(* CODESYS project Device.export

Project tree, tasks and I/O mapping:
  Device : CODESYS Control Win V3, 3S - Smart Software Solutions GmbH, version 3.5.16.0
    application Application
      libraries: Standard, * (System)
      task MainTask (cyclic, interval t#20ms, priority 1) calls PLC_PRG
      task VISU_TASK (cyclic, interval 100 ms, priority 31) calls VisuElems.Visu_Prg
      global variables Globale_Variablen
      program PLC_PRG [FBD]
      function block POU_Abbruch [ST]
      function block POU_Admin [ST]
      function block POU_Auswahltaste [ST]
      function block POU_Becheranzeige [FBD]
      function block POU_BecheranzeigeAuto [ST]
      function block POU_BecheranzeigeManuel [ST]
      function block POU_Kaffee_oder_Tee [ST]
      function block POU_KundenZaehler [ST]
      visualisation Visualisierung_Getrankeautomat
*)

// Device/Application/Globale_Variablen
{attribute 'qualified_only'}
VAR_GLOBAL
	// Variable für die Simulation der Becheranzeige
	Fuellstand: INT := 0;
	Leer: BOOL;
	Full: BOOL;
	// Eingänge
	S1:BOOL; // Kaffee
	S2:BOOL; // Tee
	S3:BOOL; // Zucker
	S4:BOOL; // Milch
	S5:BOOL; // Münzeinwurf
	S6:BOOL; // Admin
	S9:BOOL; // Abbruch
	// Anzeigen
	H1:BOOL; // Kaffee
	H2:BOOL;// Tee
	H3:INT := 0; // Zucker
	H4:INT := 0; // Milch
	H5:BOOL; // Münzeinwurf
	H6:BOOL; // Admin
	H9: BOOL ; // Abbruch
	// Variable für die "Kundenzähler"
	KundenZahl:Word;
	disp_Kundenzahl:STRING;
	// Displayvariable
	Display:STRING;
	//Verriegelungsvariablen für Milch und Zucker
	Flanke1:BOOL:=TRUE;
	Flanke2:BOOL:=TRUE;
	G1:BOOL:=TRUE;
	G2:BOOL:=True;
	// Füllsensor 
	HB2:BOOL;
	B2:BOOL;
	B1:BOOL;
	// 
	x2:BOOL;
	K1:BOOL:=TRUE;
	
	// Variable für die Dosierung Milch und Zucker
	Anzahl1:INT;
    Anzahl2:INT;
END_VAR

// Device/Application/PLC_PRG
PROGRAM PLC_PRG
VAR
	
	
	// abgelaufende Zeit
	Zeit: TIME;
	Zeitint: INT := 0;
	
	POU_Becheranzeige: POU_Becheranzeige;
	
	//POU_Kaffee_0: POU_Kaffee;
	//POU_Tee_0: POU_Tee;
	

	POU_0: POU_Kaffee_oder_Tee;
	POU_Abbruch_0: POU_Abbruch;
	POU_Becheranzeige_0: POU_Becheranzeige;
	POU_Auswahltaste_0: POU_Auswahltaste;
	POU_Admin_0: POU_Admin;
	POU_KundenZahl_0: POU_KundenZaehler;
	POU_BecheranzeigeAuto_0: POU_BecheranzeigeAuto;
	POU_BecheranzeigeManuel_0: POU_BecheranzeigeManuel;
	

END_VAR

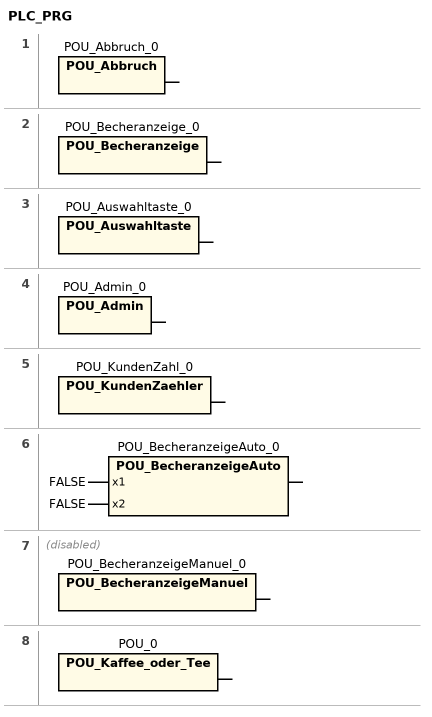
// NETWORK 1
POU_Abbruch_0(); // POU_Abbruch

// NETWORK 2
POU_Becheranzeige_0(); // POU_Becheranzeige

// NETWORK 3
POU_Auswahltaste_0(); // POU_Auswahltaste

// NETWORK 4
POU_Admin_0(); // POU_Admin

// NETWORK 5
POU_KundenZahl_0(); // POU_KundenZaehler

// NETWORK 6
POU_BecheranzeigeAuto_0(x1 := FALSE, x2 := FALSE); // POU_BecheranzeigeAuto

// NETWORK 7 (disabled)
// POU_BecheranzeigeManuel_0(); // POU_BecheranzeigeManuel

// NETWORK 8
POU_0(); // POU_Kaffee_oder_Tee

END_PROGRAM

// Device/Application/POU_Abbruch
FUNCTION_BLOCK POU_Abbruch
VAR_INPUT
END_VAR
VAR_OUTPUT
END_VAR
VAR
END_VAR

Globale_Variablen.H9:= Globale_Variablen.S9;
IF (Globale_Variablen.H9  = TRUE AND Globale_Variablen.Leer = FALSE AND Globale_Variablen.B1=FALSE )THEN
	
	Globale_Variablen.K1 := TRUE;
	Globale_Variablen.S1:= FALSE;
	Globale_Variablen.S2:= FALSE;
	Globale_Variablen.H1:= FALSE;
	Globale_Variablen.H2:= FALSE;
//Globale_Variablen.S3:= FALSE;
 //	Globale_Variablen.S4:= FALSE;
	Globale_Variablen.H3:= 0;
	Globale_Variablen.H4:= 0;
	Globale_Variablen.H5:= FALSE;
	Globale_Variablen.S5:= FALSE;
	//Globale_Variablen.H6:= FALSE;
	//Globale_Variablen.S6:= FALSE;
	Globale_Variablen.Display := 'Abbruch';
	//Globale_Variablen.H9:= TRUE;
	Globale_Variablen.Leer:=FALSE;
	Globale_Variablen.Full:=FALSE;
	Globale_Variablen.G1 := TRUE;
	
END_IF
// In der oberen If Bedingung wird gefragt ob die Abbruchtaster S9 betätig wurde , wenn ja 
// dann soll alles abgebrochen werden und Lampe H9 leuchten so lange S9 betätigt ist . 

IF Globale_Variablen.H9=FALSE THEN
		//Globale_Variablen.H9:= FALSE;
		Globale_Variablen.Display := 'Bereit';
END_IF

END_FUNCTION_BLOCK

// Device/Application/POU_Becheranzeige
FUNCTION_BLOCK POU_Becheranzeige

VAR	
	//Fuellstand: INT := 0;
	//Leer: BOOL;
	//Voll: BOOL;
END_VAR

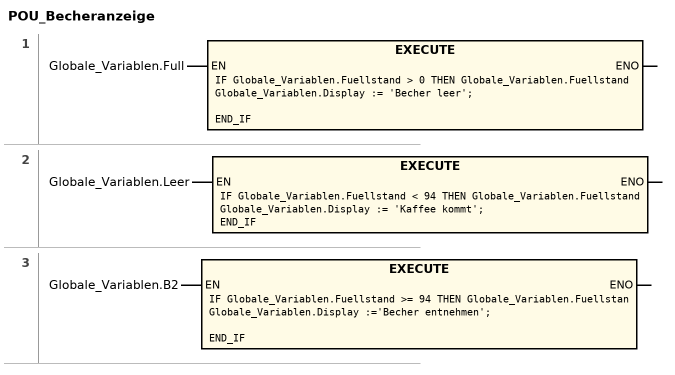
// NETWORK 1
IF Globale_Variablen.Full THEN
    IF Globale_Variablen.Fuellstand > 0 THEN Globale_Variablen.Fuellstand := 0;
    Globale_Variablen.Display := 'Becher leer';
    
    END_IF
END_IF

// NETWORK 2
IF Globale_Variablen.Leer THEN
    IF Globale_Variablen.Fuellstand < 94 THEN Globale_Variablen.Fuellstand := Globale_Variablen.Fuellstand + 1;
    Globale_Variablen.Display := 'Kaffee kommt';
    END_IF
END_IF

// NETWORK 3
IF Globale_Variablen.B2 THEN
    IF Globale_Variablen.Fuellstand >= 94 THEN Globale_Variablen.Fuellstand := 0;
    Globale_Variablen.Display :='Becher entnehmen';
    	
    END_IF
END_IF

END_FUNCTION_BLOCK

// Device/Application/POU_Auswahltaste
FUNCTION_BLOCK POU_Auswahltaste
VAR_INPUT
END_VAR
VAR_OUTPUT
END_VAR
VAR
Merker1:BOOL;
Anzahl3:INT;
Merker2:BOOL;
Anzahl4:INT;


END_VAR

// H3 Zuckeranzeige

Globale_Variablen.Flanke1 := Globale_Variablen.S3 AND NOT Merker1 ;
Merker1 := Globale_Variablen.S3;

IF Globale_Variablen.Flanke1 = 1 AND Globale_Variablen.G1=TRUE THEN 
	Anzahl3 :=Anzahl3 +1;
	Globale_Variablen.H3:=Anzahl3;
END_IF


IF Merker1 = TRUE  THEN 

IF Anzahl3 <= 3 THEN
	CASE Anzahl3 OF
      
		1: Globale_Variablen.Display := '1x Zucker'; 
		2:  Globale_Variablen.Display := '2x Zucker';
		ELSE 
			Globale_Variablen.H3 := 0;
			
 	END_CASE


END_IF
END_IF

IF (Anzahl3 >= 3 OR  Globale_Variablen.S9) THEN
	Anzahl3 := 0;
END_IF

// H4 Milchanzeige
Globale_Variablen.Flanke2 := Globale_Variablen.S4 AND NOT Merker2 AND Globale_Variablen.G1;
Merker2 := Globale_Variablen.S4;


IF Globale_Variablen.Flanke2 = 1 AND Globale_Variablen.G2=TRUE THEN 
	Anzahl4 :=Anzahl4 +1;
	Globale_Variablen.H4:=Anzahl4;
END_IF


IF Merker2 =TRUE  THEN 

IF Anzahl4 <= 3 THEN
	CASE Anzahl4 OF
      
		1: Globale_Variablen.Display := '1x Milch'; 
		2:  Globale_Variablen.Display := '2x Milch';
		ELSE 
			Globale_Variablen.H4 := 0;
			
 	END_CASE
		
END_IF
END_IF

IF (Anzahl4 >= 3 OR    Globale_Variablen.S9) THEN
	Anzahl4 := 0;
END_IF


IF (Anzahl3 >= 3 OR    Globale_Variablen.S9) THEN
	Anzahl3 := 0;
END_IF

END_FUNCTION_BLOCK

// Device/Application/POU_Admin
FUNCTION_BLOCK POU_Admin
VAR_INPUT
END_VAR
VAR_OUTPUT
END_VAR
VAR
I:INT;
x1:Bool;
Flanke1:BOOL;
Flanke2:BOOL;
Merker1:BOOL;
Merker2:BOOL;
MerkerS6:BOOL;
Merker3:BOOL;
Merker4:BOOL;
MerkerS5:BOOL;

Anzahl1:INT;
Anzahl2:INT;
END_VAR

// Globale_Variablen.H6 :=Globale_Variablen.S6;
// IF Globale_Variablen.H6 = TRUE THEN 
// 
// END_IF 
Merker3:=Globale_Variablen.H5;
 
// die Lokale Variable Merker3 dient dazu , ob die Taster S5 betätigt ist  und dementsprechend H5 leuchtet
// wenn ja , dann soll der Programm in die 2. Bedingung springen , 
//wenn nein , dann die erste If Bedingung muss ausgeführt werden
// d.h ob Münze eingeworfen ist oder nicht 

IF (Globale_Variablen.S6= TRUE AND Merker3 = FALSE) THEN 
	Globale_Variablen.H6 := TRUE;
	Globale_Variablen.H5:= FALSE;
	Globale_Variablen.Display:='Admin';

END_IF


//in der oberen If Bedingung wird geprüft welcher Taster zuerst betätigt wird, 
//genauer gesagt wenn die Lampe H6 true ist dann wird die Lampe H5 auf False gesetzt und damit blockiert.

 Merker4:=Globale_Variablen.H6;
 
IF (Globale_Variablen.S5=TRUE AND Merker4= FALSE) THEN 
	Globale_Variablen.H5:= TRUE;
	Globale_Variablen.H6:=FALSE;
	
END_IF
//in der oberen If Bedingung wird geprüft welcher Taster zuerst betätigt wird, 
//genauer gesagt wenn die  Lampe H5 true ist dann wird  die Lampe H6 auf False gesetzt und damit blockiert.
Globale_Variablen.H6:=Globale_Variablen.S6;

END_FUNCTION_BLOCK

// Device/Application/POU_KundenZaehler
FUNCTION_BLOCK POU_KundenZaehler
VAR_INPUT 
	//x1:BOOL;
	CTU:CTU;
	CV:INT;
END_VAR
VAR_OUTPUT
END_VAR
VAR
END_VAR

//x1:=(Globale_Variablen.H5= TRUE) AND (Globale_Variablen.H2=TRUE OR Globale_Variablen.H1=TRUE);
// um die Aufwand etwas erleichtern und Programm übersichtlicher zu machen haben wir uns entschieden , 
// eine lokale Variable x1 zu benutzen . X1 ist true wenn die Münze eingeworfen und eine der Getränke 
// gewählt wurde 
// x1 ist der Eingang der untenstehende "CTU" Bausteine , welche hochzählt wenn x1 true ist .

	CTU(
	CU:= (Globale_Variablen.B1 and Globale_Variablen.H5), 
	RESET:=FALSE , 
	PV:=1000 , 
	Q=> , 
	CV=> Globale_Variablen.KundenZahl);
	Globale_Variablen.disp_Kundenzahl:= ANY_TO_STRING(Globale_Variablen.KundenZahl);

END_FUNCTION_BLOCK

// Device/Application/POU_BecheranzeigeAuto
FUNCTION_BLOCK POU_BecheranzeigeAuto
VAR_INPUT
	x1:BOOL;
	x2:BOOL;
	TON:TON;
	
END_VAR
VAR_OUTPUT
END_VAR
VAR
END_VAR

IF Globale_Variablen.H5 AND (Globale_Variablen.H1 OR Globale_Variablen.H2 ) THEN
	x1:=TRUE;
	Globale_Variablen.K1:=FALSE;
	END_IF

IF Globale_Variablen.Full=TRUE THEN
	Globale_Variablen.Full:=FALSE;
	
END_IF
// In der oberen If Bedingung wird gefragt ob der Becher am Anfang der Simulation voll ist , 
//wenn ja wird es "geleert" also Becher wird entnommen .

IF Globale_Variablen.Leer=TRUE THEN
	Globale_Variablen.Leer:=FALSE;
	Globale_Variablen.B2:=FALSE;	
	
END_IF

TON(IN:=x1 , PT:=T#3S , Q=> Globale_Variablen.x2 , ET=> );

IF Globale_Variablen.x2=TRUE THEN
	Globale_Variablen.Leer:=TRUE;
	END_IF
// "Globale_Variablen.Leer " ist zuständig für Füllen des Bechers und
// ist dann True wenn in Normal (Müneinwurf) oder Admin modus eine der Getränke gewählt wurde

IF Globale_Variablen.Fuellstand = 80  THEN 
	 Globale_Variablen.S1:=FALSE;
      Globale_Variablen.S2:=FALSE;	

	    Globale_Variablen.H1:=FALSE;	
		Globale_Variablen.H2:=FALSE;
		Globale_Variablen.K1:=TRUE;
		Globale_Variablen.B1:=TRUE;	
		GLobale_Variablen.Leer:=FALSE;
		Globale_Variablen.Display:='Becher entnehmen';
	END_IF
// In der Oberen If Bedingung wird die Maximale Füllstand des Bechers geprüft und wenn es erreicht wird
// darf der Becher nicht mehr gefüllt werden
IF Globale_Variablen.K1=FALSE  THEN 
	Globale_Variablen.HB2 :=FALSE;
	Globale_Variablen.B2 :=FALSE;
END_IF

IF Globale_Variablen.HB2 =TRUE  THEN
			Globale_Variablen.Full:=True;
			Globale_Variablen.H1:= FALSE;
			Globale_Variablen.H2:= FALSE;
			Globale_Variablen.H3:= 0;
			Globale_Variablen.H4:= 0;
			Globale_Variablen.S3:= FALSE;
			Globale_Variablen.S4:= FALSE;
			Globale_Variablen.H5:= FALSE;
			Globale_Variablen.S5:=FALSE;
			Globale_Variablen.Display:='Bereit';
			Globale_Variablen.B1:=FALSE;
END_IF
Globale_Variablen.HB2:=Globale_Variablen.B2;
// In unserem Programm B2 simuliert "Becherentnahme" , wenn der Becher entnommen wurde , 
// muss alle vorher gewählte Variable auf Anfangszustand zurückgesetzt werden .


// ADMIN MODUS BECHERANZEIGE

 IF Globale_Variablen.H6 AND (Globale_Variablen.S1 OR Globale_Variablen.S2) THEN 
	 Globale_Variablen.Leer:= True;
 END_IF
// "Globale_Variablen.Leer " ist zuständig für Füllen des Bechers und
// ist dann True wenn in Normal (Müneinwurf) oder Admin modus eine der Getränke gewählt wurde

IF Globale_Variablen.Full=TRUE THEN
	Globale_Variablen.Full:=FALSE;
	
END_IF
// In der oberen If Bedingung wird gefragt ob der Becher am Anfang der Simulation voll ist , 
//wenn ja wird es "geleert" also Becher wird entnommen .


IF Globale_Variablen.Fuellstand =80 THEN 
	Globale_Variablen.Leer:= FALSE;
END_IF
// In der Oberen If Bedingung wird die Maximale Füllstand des Bechers geprüft und wenn es erreicht wird
// darf der Becher nicht mehr gefüllt werden

IF Globale_Variablen.HB2 =TRUE THEN
			Globale_Variablen.Full:=True;
			Globale_Variablen.H1:= FALSE;
			Globale_Variablen.H2:= FALSE;
			Globale_Variablen.Anzahl1 := 0;
			Globale_Variablen.Anzahl2 := 0;
			Globale_Variablen.H3:= 0;
			Globale_Variablen.H4:= 0;
			Globale_Variablen.S3:= FALSE;
			Globale_Variablen.S4:= FALSE;
			Globale_Variablen.H5:= FALSE;
			Globale_Variablen.S5:=FALSE;
			Globale_Variablen.H3:= 0;
			Globale_Variablen.H4:= 0;
			Globale_Variablen.B1:=FALSE;
			Globale_Variablen.Fuellstand :=0;
			
			Globale_Variablen.G1:= TRUE;

		END_IF




IF Globale_Variablen.H5=TRUE THEN 
	Globale_Variablen.S3:= FALSE;
		Globale_Variablen.S6:= FALSE;
	Globale_Variablen.S4:= FALSE;
	Globale_Variablen.Flanke1:= FALSE;
	Globale_Variablen.G1 := FALSE;
	
END_IF


// In unserem Programm B2 simuliert "Becherentnahme" , wenn der Becher entnommen wurde , 
// muss alle vorher gewählte Variable auf Anfangszustand zurückgesetzt werden .

END_FUNCTION_BLOCK

// Device/Application/POU_BecheranzeigeManuel
FUNCTION_BLOCK POU_BecheranzeigeManuel
VAR_INPUT
END_VAR
VAR_OUTPUT
END_VAR
VAR
END_VAR

Globale_Variablen.Leer:=Globale_Variablen.S6 AND (Globale_Variablen.S1 OR Globale_Variablen.S2);
// "Globale_Variablen.Leer " ist zuständig für Füllen des Bechers und
// ist dann True wenn in Normal (Müneinwurf) oder Admin modus eine der Getränke gewählt wurde

IF Globale_Variablen.Full=TRUE THEN
	Globale_Variablen.Full:=FALSE;
	
END_IF
// In der oberen If Bedingung wird gefragt ob der Becher am Anfang der Simulation voll ist , 
//wenn ja wird es "geleert" also Becher wird entnommen .


IF Globale_Variablen.Fuellstand =80 THEN 
	Globale_Variablen.Leer:= FALSE;
END_IF
// In der Oberen If Bedingung wird die Maximale Füllstand des Bechers geprüft und wenn es erreicht wird
// darf der Becher nicht mehr gefüllt werden

IF Globale_Variablen.B2 =TRUE THEN
			Globale_Variablen.Full:=True;
			Globale_Variablen.H1:= FALSE;
			Globale_Variablen.H2:= FALSE;
			Globale_Variablen.H3:= 0;
			Globale_Variablen.H4:= 0;
			Globale_Variablen.S3:= FALSE;
			Globale_Variablen.S4:= FALSE;
			Globale_Variablen.H5:= FALSE;
			Globale_Variablen.S5:=FALSE;
			Globale_Variablen.Display:='Bereit';
			Globale_Variablen.B1:=FALSE;
			Globale_Variablen.Fuellstand :=0;

		END_IF
		
// In unserem Programm B2 simuliert "Becherentnahme" , wenn der Becher entnommen wurde , 
// muss alle vorher gewählte Variable auf Anfangszustand zurückgesetzt werden .

END_FUNCTION_BLOCK

// Device/Application/POU_Kaffee_oder_Tee
FUNCTION_BLOCK POU_Kaffee_oder_Tee
VAR_INPUT 

	Merker1:BOOL;
	Merker2:BOOL;
END_VAR
VAR_OUTPUT
END_VAR
VAR
END_VAR


 Merker2:=Globale_Variablen.H2;
// die Lokale Variable Merker2 dient dazu , ob die Taster S2 betätigt ist  und dementsprechend H2 leuchtet
// wenn ja , dann soll der Programm in die 2. Bedingung springen , 
//wenn nein , dann die erste If Bedingung muss ausgeführt werden

IF (Globale_Variablen.S1=TRUE AND  Merker2 = FALSE AND Globale_Variablen.H5) THEN 
	Globale_Variablen.H1 := TRUE;
	Globale_Variablen.S2:= FALSE;
	

END_IF


IF Globale_Variablen.H1 = TRUE THEN 
	Globale_Variablen.Display:='Kaffee kommt';
END_IF
//in der oberen If Bedingung wird geprüft welcher Taster zuerst betätigt wird, 
//genauer gesagt wenn der taster S1 true ist dann wird der Taster S2 auf False gesetzt und damit blockiert.




 Merker1:=Globale_Variablen.H1;
IF (Globale_Variablen.S2 AND Merker1 = FALSE and Globale_Variablen.H5 ) THEN 
	Globale_Variablen.H2 := TRUE;
	Globale_Variablen.S1:=FALSE;
	
END_IF
IF Globale_Variablen.H2 = TRUE THEN 
	Globale_Variablen.Display:='Tee kommt';
END_IF
//in der oberen If Bedingung wird geprüft welcher Taster zuerst betätigt wird, 
//genauer gesagt wenn der taster S2 true ist dann wird der Taster S1 auf False gesetzt und damit blockiert.

//Globale_Variablen.H5:= Globale_Variablen.S5;

END_FUNCTION_BLOCK

// Device/Application/Visualisierung_Getrankeautomat
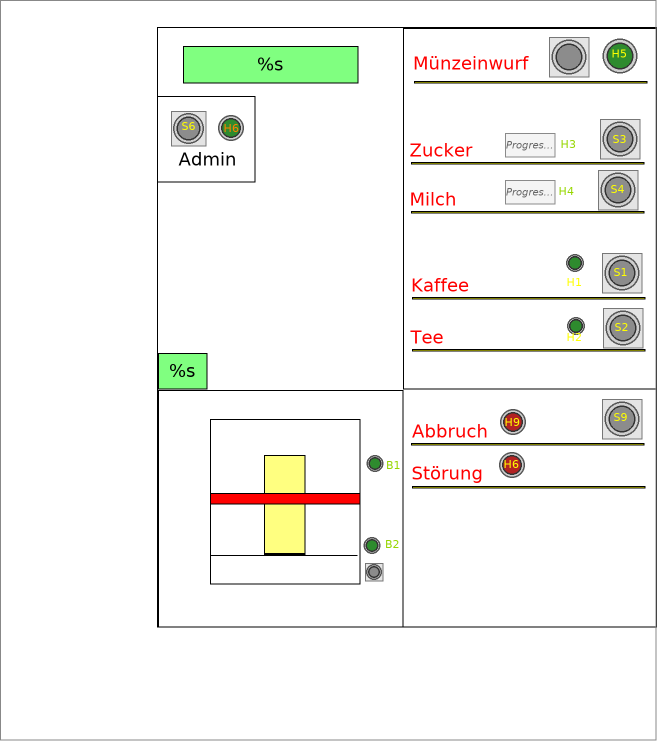
VISUALIZATION Visualisierung_Getrankeautomat  // 657x741
    Rectangle (157,27 500x600)
    Rectangle (403,28 253x361)
    PushSwitch (602,253 40x40), variable: Globale_Variablen.S1, behaviour: TAP, style: Switch-PushSwitch-Gray
    PushSwitch (603,308 40x40), variable: Globale_Variablen.S2, behaviour: TAP, style: Switch-PushSwitch-Gray
    PushSwitch (600,119 40x40), variable: Globale_Variablen.S3, behaviour: TAP, style: Switch-PushSwitch-Gray
    PushSwitch (598,170 40x40), variable: Globale_Variablen.S4, behaviour: TAP, style: Switch-PushSwitch-Gray
    Lamp1 (565,253 20x20), tooltip "Test", variable: Globale_Variablen.H1, style: Lamp-Lamp1-Green
    Lamp1 (566,306 20x40), variable: Globale_Variablen.H2, style: Lamp-Lamp1-Green
    Lamp1 (600,36 40x40), variable: Globale_Variablen.H5, style: Lamp-Lamp1-Green
    Label (414,54 114x19), "Münzeinwurf"
    Label (383,276 114x19), "Kaffee"
    Label (370,328 114x19), "Tee"
    Label (384,141 114x19), "Zucker"
    Label (376,190 114x19), "Milch"
    Label (393,422 114x19), "Abbruch"
    Label (392,465 111x17), "Störung"
    PushSwitch (602,399 40x40), variable: Globale_Variablen.S9, behaviour: TAP, style: Switch-PushSwitch-Gray
    Lamp1 (498,407 30x30), variable: Globale_Variablen.H9, style: Lamp-Lamp1-Red
    Lamp1 (497,450 30x30), style: Lamp-Lamp1-Red
    Rectangle (158,390 245x237)
    Rectangle (210,419 150x165)
    Line (211,555) (357,555)
    Label (550,44 37x23)
    Label (602,261 37x23), "S1"
    Label (603,316 37x23), "S2"
    Label (601,128 37x23), "S3"
    Label (599,178 37x23), "S4"
    Label (602,405 37x25), "S9"
    Label (601,40 37x28), "H5"
    Label (556,271 37x23), "H1"
    Label (556,326 37x23), "H2"
    Label (550,133 37x23), "H3"
    Label (548,180 37x23), "H4"
    Label (494,411 37x23), "H9"
    Label (493,453 37x23), "H6"
    Label (374,533 37x23), "B2"
    Label (375,454 37x23), "B1"
    Label (568,718 37x23)
    Progressbar (505,133 50x24), variable: Globale_Variablen.H3
    Progressbar (505,180 50x24), variable: Globale_Variablen.H4
    Rectangle (264,455 41x100)
    Rectangle (264,553 41x1)
        p1126004900: - Globale_Variablen.Fuellstand
    Rectangle (183,46 175x37), "%s", text variable: Globale_Variablen.Display
    Rectangle (414,81 233x2)
    Rectangle (411,211 233x2)
    Rectangle (411,443 233x2)
    Rectangle (412,486 233x2)
    Rectangle (412,297 233x2)
    Rectangle (157,96 98x86)
    Rectangle (412,349 233x2)
    Rectangle (411,162 233x2)
    Label (168,151 79x17), "Admin"
    Lamp1 (216,113 30x30), variable: Globale_Variablen.H6, style: Lamp-Lamp1-Green
    PushSwitch (171,111 35x35), variable: Globale_Variablen.S6, behaviour: TOGGLE, style: Switch-PushSwitch-Gray
    Label (170,115 37x23), "S6"
    Label (213,117 37x23), "H6"
    Rectangle (158,353 49x36), "%s", text variable: Globale_Variablen.disp_Kundenzahl
    Lamp1 (365,454 20x19), variable: Globale_Variablen.B1, style: Lamp-Lamp1-Green
    Lamp1 (362,536 20x19), variable: Globale_Variablen.HB2, style: Lamp-Lamp1-Green
    PushSwitch (364,563 20x18), variable: Globale_Variablen.B2, behaviour: TAP, style: Switch-PushSwitch-Gray
    Rectangle (210,493 150x11), invisible if: Globale_Variablen.K1
    Label (547,43 37x22)
    PushSwitch (549,37 40x40), variable: Globale_Variablen.S5, behaviour: TAP, style: Switch-PushSwitch-Gray
END_VISUALIZATION
